FUNCTION_BLOCK FB_Motor1
VAR_INPUT
	new: BOOL;
	pos: REAL;
	vel: REAL;
	acc: REAL;
	dec: REAL;
END_VAR
VAR_OUTPUT
END_VAR
VAR
	will_new: BOOL;
	will_pos: REAL;
	will_vel: REAL;
	will_acc: REAL;
	will_dec: REAL;
	state: E_MoveState;
	PowerAxis: MC_Power;
	PowerAxisOut: ST_McOutputs;
	MoveAxis: MC_MoveAbsolute;
	MoveAbsoluteOut: ST_McOutputs;
	Reset: MC_Reset;
	ResetOut: ST_McOutputs;
END_VAR

GVL_IO.AxisRef1();

IF new THEN
	will_new := TRUE;
	will_pos := pos;
	will_vel := vel;
	will_acc := acc;
	will_dec := dec;
END_IF

CASE state OF
	E_MoveState.init:
		MoveAxis.Execute := FALSE;
		Reset.Execute := FALSE;
		state := E_MoveState.enable;
	E_MoveState.enable:
		PowerAxis.Enable := TRUE;
		PowerAxis.Enable_Positive := TRUE;
		PowerAxis.Enable_Negative := TRUE;
		IF PowerAxis.Status THEN
			state := E_MoveState.forward;
		ELSIF PowerAxis.Error THEN
			state := E_MoveState.error;
		END_IF
	E_MoveState.forward:
		IF will_new THEN
			MoveAxis.Position := will_pos;
			MoveAxis.Velocity := will_vel;
			MoveAxis.Acceleration := will_acc;
			MoveAxis.Deceleration := will_dec;
			MoveAxis.BufferMode := MC_Buffered;
			MoveAxis.Execute := TRUE;
			will_new := FALSE;
		ELSE
			MoveAxis.Execute := FALSE;
		END_IF
		(**IF MoveAxis1.Active THEN
			MoveAxis1.Execute := FALSE;
			state := E_MoveState.new_target_position;
		ELSIF MoveAxis1.CommandAborted OR MoveAxis1.Error THEN
			state := E_MoveState.error;
		END_IF*)
	E_MoveState.error:
		IF GVL_IO.AxisRef1.Status.Error THEN
			state := E_MoveState.reset;
		ELSE
			state := E_MoveState.init;
		END_IF
	E_MoveState.reset:
		Reset.Execute := TRUE;
		IF Reset.Done THEN
			state := E_MoveState.init;
		ELSIF Reset.Error THEN
			state := E_MoveState.init;
		END_IF
END_CASE

ACT_Power();
ACT_Move();
ACT_Reset();

ACTION ACT_Move:
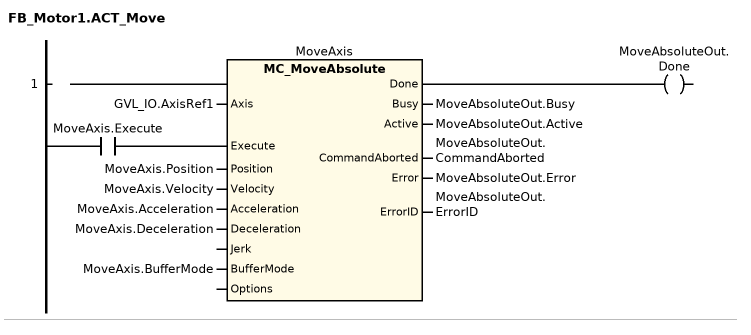
// NETWORK 1
MoveAxis(
    Axis := GVL_IO.AxisRef1,
    Execute := MoveAxis.Execute,
    Position := MoveAxis.Position,
    Velocity := MoveAxis.Velocity,
    Acceleration := MoveAxis.Acceleration,
    Deceleration := MoveAxis.Deceleration,
    BufferMode := MoveAxis.BufferMode,
    Busy => MoveAbsoluteOut.Busy,
    Active => MoveAbsoluteOut.Active,
    CommandAborted => MoveAbsoluteOut.CommandAborted,
    Error => MoveAbsoluteOut.Error,
    ErrorID => MoveAbsoluteOut.ErrorID); // MC_MoveAbsolute
MoveAbsoluteOut.Done := MoveAxis.Done;
END_ACTION

ACTION ACT_Power:
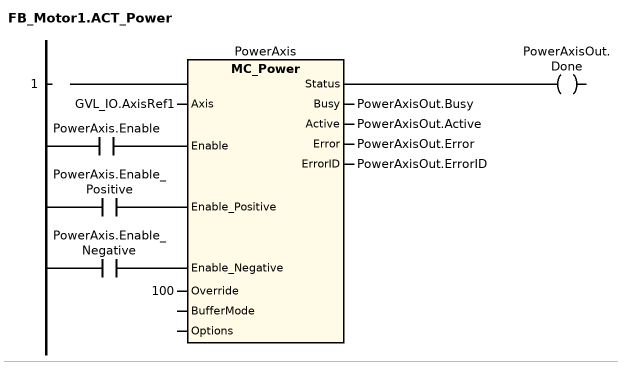
// NETWORK 1
PowerAxis(
    Axis := GVL_IO.AxisRef1,
    Enable := PowerAxis.Enable,
    Enable_Positive := PowerAxis.Enable_Positive,
    Enable_Negative := PowerAxis.Enable_Negative,
    Override := 100,
    Busy => PowerAxisOut.Busy,
    Active => PowerAxisOut.Active,
    Error => PowerAxisOut.Error,
    ErrorID => PowerAxisOut.ErrorID); // MC_Power
PowerAxisOut.Done := PowerAxis.Status;
END_ACTION

ACTION ACT_Reset:
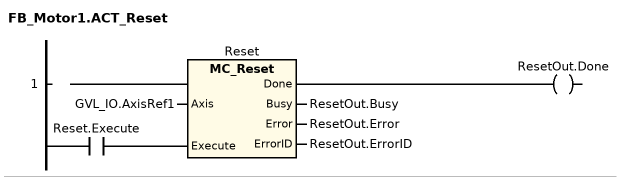
// NETWORK 1
Reset(
    Axis := GVL_IO.AxisRef1,
    Execute := Reset.Execute,
    Busy => ResetOut.Busy,
    Error => ResetOut.Error,
    ErrorID => ResetOut.ErrorID); // MC_Reset
ResetOut.Done := Reset.Done;
END_ACTION

END_FUNCTION_BLOCK

(* stored: Version 1.1.0.1, ProductVersion 3.1.4024.11
   POU FB_Motor1: Id {8ab050cb-81c0-4d6c-8777-1347a3f16775}, SpecialFunc None
   Action ACT_Move: Id {1ed9d3a1-4079-440c-b1d1-80cc1bf80bd7}
   Action ACT_Power: Id {2ebad139-5492-4334-805e-0a70420b761e}
   Action ACT_Reset: Id {8c85953c-dcad-4548-ac89-7bc9c4add938} *)
